// TwinCAT 3 PLC project PLC
// ProgramVersion: 3.1.4024.0
// libraries:
//   EfficientIO Communicator, * (EfficientIO)
//   EfficientIO Energy Basic, * (EfficientIO)
//   Lynus Energy ModbusRTU, * (Lynus AG)
//   Lynus HTTP Functions, * (Lynus AG)
//   Lynus Persistent Data V1, * (Lynus AG)
//   Lynus Standards, * (EfficientIO)
//   Tc2_Math, * (Beckhoff Automation GmbH)
//   Tc2_MBus, * (Beckhoff Automation GmbH)
//   Tc2_ModbusRTU, * (Beckhoff Automation GmbH)
//   Tc2_SerialCom, * (Beckhoff Automation GmbH)
//   Tc2_Standard, * (Beckhoff Automation GmbH)
//   Tc2_System, * (Beckhoff Automation GmbH)
//   Tc2_TcpIp, * (Beckhoff Automation GmbH)
//   Tc2_Utilities, * (Beckhoff Automation GmbH)
//   Tc3_IotBase, * (Beckhoff Automation GmbH)
//   Tc3_JsonXml, * (Beckhoff Automation GmbH)
//   Tc3_Module, * (Beckhoff Automation GmbH)
//   VModbusBase, * (VSA GmbH)
//   VModbusTcp, * (VSA GmbH)
// project tree:
//   / FastTask.TcTTO, MiddleTask.TcTTO, SlowTask.TcTTO
//   FB/ FB_Delta_PV_Inverter_Sunspec.TcPOU (not stored) (excluded from build), FB_Hoval.TcPOU, FB_KL6xxx_ModbusRTU_22B_Master.TcPOU (excluded from build), FB_ShellyHT_Udp.TcPOU, FB_Shelly_3EM.TcPOU (not stored) (excluded from build), FB_Shelly_HT.TcPOU (excluded from build), FB_Shelly_3EM_Helper.TcPOU (not stored) (excluded from build), FB_Shelly_HTplus.TcPOU (excluded from build), FB_Shelly_HT_Helper.TcPOU (not stored) (excluded from build), FB_Shelly_HTplus_Helper.TcPOU (excluded from build), FB_Shelly_Pro.TcPOU (excluded from build), FB_Shelly_Pro3EM.TcPOU, FB_Shelly_Pro3EM_Helper.TcPOU (not stored)
//   POUs/ prgComEffIO.TcPOU, prgEM.TcPOU, prgGrid.TcPOU (not stored), prgHeizen.TcPOU, prgHouse.TcPOU, prgMBUS.TcPOU, prgPersistent.TcPOU, prgPV.TcPOU, prgRWEffIO.TcPOU (not stored), prgSmartMe.TcPOU, prgVarEffIO.TcPOU (not stored)
// real-time tasks:
//   TASK FastTask: cycle T#5ms, priority 19, ADS port 351
//   TASK SlowTask: cycle T#20ms, priority 21, ADS port 352
//   TASK MiddleTask: cycle T#10ms, priority 20, ADS port 353
// I/O:
//   DEVICE Gerät 2 (CX-BK)
//     Box 1 (CX-BK)
//   DEVICE Device 1 (Beckhoff CCAT)
//   DEVICE Device 3 (RT-Ethernet Protocol), AmsNetId 5.123.218.205.4.1
//     Box 2 (BK9050)
// variable links:
//   PLC/PLC Instance <-> Device 2 (CX-BK)/Box 1 (CX-BK)
//     FastTask Inputs/prgMBUS.stComIn @bit {16..184 step 8} <-> Term 2 (KL6781)/Channel 1/Data In {0..21}  (22 links)
//     FastTask Inputs/prgMBUS.stComIn <-> Term 2 (KL6781)/Channel 1/Status
//     FastTask Outputs/prgMBUS.stComOut <-> Term 2 (KL6781)/Channel 1/Ctrl
//     FastTask Outputs/prgMBUS.stComOut @bit {16..184 step 8} <-> Term 2 (KL6781)/Channel 1/Data Out {0..21}  (22 links)
//     MiddleTask Inputs/prgGrid.fbGrid.fbKL3403.byStateCH1 <-> Term 5 (KL3403)/Channel 1/Status
//     MiddleTask Inputs/prgGrid.fbGrid.fbKL3403.byStateCH2 <-> Term 5 (KL3403)/Channel 2/Status
//     MiddleTask Inputs/prgGrid.fbGrid.fbKL3403.byStateCH3 <-> Term 5 (KL3403)/Channel 3/Status
//     MiddleTask Inputs/prgGrid.fbGrid.fbKL3403.iDataInCH1 <-> Term 5 (KL3403)/Channel 1/Daten Ein
//     MiddleTask Inputs/prgGrid.fbGrid.fbKL3403.iDataInCH2 <-> Term 5 (KL3403)/Channel 2/Daten Ein
//     MiddleTask Inputs/prgGrid.fbGrid.fbKL3403.iDataInCH3 <-> Term 5 (KL3403)/Channel 3/Daten Ein
//     MiddleTask Inputs/prgGrid.fbKBusState.uiKBusState_OUT <-> Inputs/State
//     MiddleTask Outputs/prgGrid.fbGrid.fbKL3403.byCntrCH1 <-> Term 5 (KL3403)/Channel 1/Kontrolle
//     MiddleTask Outputs/prgGrid.fbGrid.fbKL3403.byCntrCH2 <-> Term 5 (KL3403)/Channel 2/Kontrolle
//     MiddleTask Outputs/prgGrid.fbGrid.fbKL3403.byCntrCH3 <-> Term 5 (KL3403)/Channel 3/Kontrolle
//   PLC/PLC Instance <-> Device 3 (RT-Ethernet Protocol)/Box 2 (BK9050)
//     FastTask Inputs/prgPV.fb_RTU_Master.fbmodbusmaster.InData @bit {16..184 step 8} <-> Term 4 (KL6041)/Channel 1/Data In {0..21}  (22 links)
//     FastTask Inputs/prgPV.fb_RTU_Master.fbmodbusmaster.InData <-> Term 4 (KL6041)/Channel 1/State
//     FastTask Outputs/prgPV.fb_RTU_Master.fbmodbusmaster.OutData <-> Term 4 (KL6041)/Channel 1/Ctrl
//     FastTask Outputs/prgPV.fb_RTU_Master.fbmodbusmaster.OutData @bit {16..184 step 8} <-> Term 4 (KL6041)/Channel 1/Data Out {0..21}  (22 links)

CONFIGURATION PLC
    RESOURCE PLC ON TwinCAT3
        TASK FastTask(INTERVAL := T#5ms, PRIORITY := 19);
        TASK MiddleTask(INTERVAL := T#10ms, PRIORITY := 20);
        TASK SlowTask(INTERVAL := T#20ms, PRIORITY := 21);
        PROGRAM prgRWEffIO WITH FastTask : prgRWEffIO;
        PROGRAM prgVarEffIO WITH FastTask : prgVarEffIO;
        PROGRAM prgPV WITH FastTask : prgPV;
        PROGRAM prgMBUS WITH FastTask : prgMBUS;
        PROGRAM prgPersistent WITH MiddleTask : prgPersistent;
        PROGRAM prgGrid WITH MiddleTask : prgGrid;
        PROGRAM prgHouse WITH MiddleTask : prgHouse;
        PROGRAM prgEM WITH MiddleTask : prgEM;
        PROGRAM prgSmartMe WITH MiddleTask : prgSmartMe;
        PROGRAM prgHeizen WITH MiddleTask : prgHeizen;
        PROGRAM prgComEffIO WITH SlowTask : prgComEffIO;
    END_RESOURCE
END_CONFIGURATION

// ---- POUs/prgPV.TcPOU
PROGRAM prgPV
VAR
	lrPower_PV1					: LREAL;								//{#lynus.ag#()}
	lrPower_PV2					: LREAL;								//{#lynus.ag#()}
	lrPower_PV3					: LREAL;								//{#lynus.ag#()}
	fb_PV_1						: FB_delta_PV_inverter_sunspec;
	fb_PV_2						: FB_delta_PV_inverter_sunspec;
	fb_PV_3						: FB_delta_PV_inverter_sunspec;

	fb_RTU_Master 				: FB_KL6xxx_ModbusRTU_22B_Master;
	fbModbusRtuMaster_KL6x22B	: ModbusRtuMaster_KL6x22B;
	uint_KBusState				: UINT;							//{#lynus.ag#()}
	fbConfigKL6041 				: KL6Configuration;
	mExecute					: BOOL:= FALSE;
	int_Handshake				: INT:=0;
	mode						: ComSerialLineMode_t:=2;	
	wArrayReceiveBuffer			: ARRAY[0..130] OF WORD;
	lrCounterPV1				: LREAL;				//{#lynus.ag#()}
	lrCounterPV2				: LREAL;				//{#lynus.ag#()}
	lrCounterPV3				: LREAL;				//{#lynus.ag#()}
	rHeatSinkTemp_PV1			: REAL;					//{#lynus.ag#()}
	rHeatSinkTemp_PV2			: REAL;					//{#lynus.ag#()}
	rHeatSinkTemp_PV3			: REAL;					//{#lynus.ag#()}
	rCabinetTemp_PV1			: REAL;					//{#lynus.ag#()}
	rCabinetTemp_PV2			: REAL;					//{#lynus.ag#()}
	rCabinetTemp_PV3			: REAL;					//{#lynus.ag#()}
	usiAddress					: BYTE;
	usi_ScannedAddress			: REAL;
	
END_VAR


fb_RTU_Master(
	bConfigTerminal:= TRUE, 
	uiKBusState_IN:= uint_KBusState, 
	bBusy=> , 
	byErrorWarning=> , 
	byActualAdressInUse=> , 
	diNrOfMBRTUMasterLine_OUT=> , 
	eMessageMBRTUMaster=> , 
	bTerminalIsConfigured=> );

fb_PV_1(
	bEnable:= TRUE, 
	byMBAdress:=2 , 
	diNrOfMBRTUMasterLine_IN:= fb_RTU_Master.diNrOfMBRTUMasterLine_OUT, 
	stDeltaInverterData=> , 
	stDataEMPower_PV=> , 
	stDataEMCounter_PV=> , 
	diNrOfEM_OUT_PV=> );
fb_PV_2(
	bEnable:= TRUE, 
	byMBAdress:=3 , 
	diNrOfMBRTUMasterLine_IN:= fb_RTU_Master.diNrOfMBRTUMasterLine_OUT, 
	stDeltaInverterData=> , 
	stDataEMPower_PV=> , 
	stDataEMCounter_PV=> , 
	diNrOfEM_OUT_PV=> );
fb_PV_3(
	bEnable:= true, 
	byMBAdress:=4 , 
	diNrOfMBRTUMasterLine_IN:= fb_RTU_Master.diNrOfMBRTUMasterLine_OUT, 
	stDeltaInverterData=> , 
	stDataEMPower_PV=> , 
	stDataEMCounter_PV=> , 
	diNrOfEM_OUT_PV=> );
lrPower_PV1 		:=fb_PV_1.stDataEMPower_PV.lrPowerTotal;
lrPower_PV2 		:=fb_PV_2.stDataEMPower_PV.lrPowerTotal;
lrPower_PV3 		:=fb_PV_3.stDataEMPower_PV.lrPowerTotal;
lrCounterPV1 		:= fb_PV_1.stDataEMCounter_PV.lrCounterEnergyT1_Production;
lrCounterPV2 		:= fb_PV_2.stDataEMCounter_PV.lrCounterEnergyT1_Production;
lrCounterPV3 		:= fb_PV_3.stDataEMCounter_PV.lrCounterEnergyT1_Production;
rHeatSinkTemp_PV1	:= fb_PV_1.stDeltaInverterData.rHeatSinkTemp;
rHeatSinkTemp_PV2	:= fb_PV_2.stDeltaInverterData.rHeatSinkTemp;
rHeatSinkTemp_PV3	:= fb_PV_3.stDeltaInverterData.rHeatSinkTemp;
rCabinetTemp_PV1	:= fb_PV_1.stDeltaInverterData.rCabinetTemp;
rCabinetTemp_PV2	:= fb_PV_2.stDeltaInverterData.rCabinetTemp;
rCabinetTemp_PV3	:= fb_PV_3.stDeltaInverterData.rCabinetTemp;

(*
fbModbusRtuMaster_KL6x22B.ReadRegs(
	UnitID		:=2,
	Quantity	:=10,
	MBAddr		:=0,
	cbLength	:=20,
	pMemoryAddr	:= ADR(wArrayReceiveBuffer),
	Execute		:= TRUE,
	Timeout		:=t#1s,
	BUSY		=>,
	Error		=>,
	ErrorId		=>,
	cbRead		=>
);


fbModbusRtuMaster_KL6x22B.Execute := FALSE;

FOR usiAddress := 1 TO 247 DO
   fbModbusRtuMaster_KL6x22B.ReadRegs(UnitID := usiAddress, Execute := TRUE);
   IF NOT fbModbusRtuMaster_KL6x22B.Error THEN
      usi_ScannedAddress := usiAddress;
      EXIT;
   END_IF;
END_FOR;


// necessary for KL6041 to write the com settings
fbConfigKL6041(
	Execute 		:= mExecute,
	Mode 			:= mode,
	Baudrate 		:= 19200,
	NoDatabits 		:= 8,
	Parity 			:= 0,
	Stopbits 		:= 1,
	Handshake  		:= RS485_HALFDUPLEX, //int_Handshake,
	ContinousMode 	:= FALSE,
	pComIn 			:= ADR(fbModbusRtuMaster_KL6x22B.InData),
	pComOut 		:= ADR(fbModbusRtuMaster_KL6x22B.OutData),
	SizeComIn 		:= SIZEOF(fbModbusRtuMaster_KL6x22B.InData)		//fbModbusRtuMaster_KL6x22B
); *)

END_PROGRAM

// ---- FB/FB_KL6xxx_ModbusRTU_22B_Master.TcPOU
FUNCTION_BLOCK FB_KL6xxx_ModbusRTU_22B_Master
VAR_INPUT
	bConfigTerminal							: BOOL;																		//Possibility to configure the Terminal manually (Its only possible when the Terminal is not configured successfully)
	uiKBusState_IN							: UINT;																		//K-Bus State from the K-Bus Box on wich the Terminal is connected. (Connect with FB_K_Bus_state)
END_VAR
VAR_OUTPUT
	bBusy									: BOOL;																		//Function is Busy
	byErrorWarning							: BYTE;																		//Error Warning State
	byActualAdressInUse						: BYTE;																		//Actual Modbus Adress in Use
	diNrOfMBRTUMasterLine_OUT				: DINT;																		//Active Number from the RTU Master Function for using on other functions
	eMessageMBRTUMaster						: E_Message_MBRTUMaster;													//Message from the RTU Master Function
END_VAR				
VAR_OUTPUT PERSISTENT
	bTerminalIsConfigured					: BOOL;																		//Its True when the configuration is successfully
END_VAR
VAR		
	config_execute							: BOOL ;
	//{attribute 'hide'}
	fbKL6xxxConfig							: KL6configuration;															//FB KL6xxx to config the terminal
	fbmodbusmaster							: ModbusRtuMaster_KL6x22B;													//FB Modbus RTU
	{attribute 'hide'}
	fbmodbusmaster_Init						: ModbusRtuMaster_KL6x22B;													//FB Modbus RTU Master for workaroud regarding the internal Beckhoff problem in this function
	{attribute 'hide'}
	fbNumberDevice							: FB_NumberOfDevice;														//Function block to calcualte the number of the Device	
	{attribute 'hide'}
	fbModbusRTUMessage						: FB_MBRTUMaster_Messages;													//Modbus RTU Messages	
	{attribute 'hide'}
	FPConfigManual							: R_TRIG;																	//Internal positive Edge
	{attribute 'hide'}
	FPConfigAuto							: R_TRIG;																	//Internal positive Edge
	{attribute 'hide'}
	FPProcessCompleted						: R_TRIG;																	//Internal positive Edge
	{attribute 'hide'}
	FPError									: R_TRIG;																	//Internal positive Edge
	{attribute 'hide'}
	FPErrorIsActive							: R_TRIG;																	//Internal positive Edge
	{attribute 'hide'}
	FNInitSmall								: F_TRIG;																	//Internal negative Edge
	{attribute 'hide'}
	FNBusy									: F_TRIG;																	//Internal negative Edge
	{attribute 'hide'}
	timInit									: TON;																		//Delay to start the Terminal Configuration after the start from the plc
	{attribute 'hide'}
	timTimout								: TON;																		//Timer Timout to go on next Modbus Adress when the Ack is not set back to False
	{attribute 'hide'}
	timDissableFunctions					: TON;																		//Timer to dissable the Function after Lynus_Standards.Constants_General.tTimeDissableLynusFunctions Days without connection to the Lynus Cloud
	{attribute 'hide'}
	timResetConnectionOnGVL					: TON;																		//Timer to try reset the connection Flag on the GVL. (When somebody delete the Connection Function and make only a onlinechange)
	{attribute 'hide'}
	arrPD									: ARRAY[1..2] OF FB_PersistentData_Number;									//Function to save persistent data
	{attribute 'hide'}
	bTakeActualAdress						: BOOL;																		//True if the Current address is to be used
	{attribute 'hide'}
	bAdressHasChanged						: BOOL;																		//True if the Adress has changed
	{attribute 'hide'}
	bErrorIsActive							: BOOL;																		//True if a Error is happend. False after the next successfully read or write command
	{attribute 'hide'}
	bStopReadWrite							: BOOL;																		//Stop Function because Modbus Adress has chaged
	{attribute 'hide'}
	byLPSmallestAdress						: BYTE;																		//Loop to find out the smallest Modbus Adress
	{attribute 'hide'}
	byLPBiggestAdress						: BYTE;																		//Loop to find out the biggest Modbus Adress
	{attribute 'hide'}
	byLPActualAdress						: BYTE;																		//Loop to find out the next actuall adress
	{attribute 'hide'}
	byLPNumbersOfTotalSlaves				: BYTE;																		//Loop to find out the number of total Modbus Slaves
	{attribute 'hide'}
	bySmallestAdress						: BYTE;																		//Smallest Modbus Adress
	{attribute 'hide'}
	byBiggestAdress							: BYTE;																		//Biggest Modbus Adress
	{attribute 'hide'}
	byActualAdressInUse_CP					: BYTE;																		//Actual Modbus Adress in Use to compare it with the old one
	{attribute 'hide'}
	byNumberOfTotalSlaves					: BYTE;																		//Number of all Modbus Slaves
	{attribute 'hide'}
	byWaitInStep							: BYTE;																		//Wait in Step before start to clean data on PLC
	{attribute 'hide'}
	byLPMBAdress							: BYTE;																		//Loop for manage new Modbus Adress List after a change
	{attribute 'hide'}
	bySearchMBAdress						: BYTE;																		//Search Modbus Adress after change
	{attribute 'hide'}
	byPosInArrayMBAdress					: BYTE;																		//Save new Range from Modbus adress in the Array after a change
	{attribute 'hide'}
	iStateGVLData							: INT;																		//State machine to handle the data on the GVL
	{attribute 'hide'}
	iStateSetMBAdress						: INT;																		//State machin eto order the Modbus Adress after a change
	{attribute 'hide'}
	diCounterForGVL							: DINT;																		//Counter to clean old data on GVL
	{attribute 'hide'}
	arrRead									: ARRAY[1..Constants_Bussystems.wQuantityOfRegistersMBRTUMaster] OF WORD;	//Puffer for read out data
	{attribute 'hide'}
	arrMBAdress								: ARRAY[1..247] OF BYTE;													//Array with the actual Modbus Adress Config
END_VAR
VAR PERSISTENT
	{attribute 'conditionalshow'}
	eDeviceType								: E_MBRTUMaster_DeviceType;													//Device Type on witch the Terminal is configured
END_VAR

//Creator : Kai Ebensperger
//Company : Lynus AG
//Date : 08.07.2021
//Version : 1.0.0.0

//With this FB a serial 22 byte terminal can be configured and data can be sent/received via Modbus RTU.
//Only devices of the same type may be operated on the same master (because its not good to write to much new configurations on the terminal).
//The 1 slave that is called before the master FB in the PLC code configures the terminal
//The block must be called in a task of 5MS
//The system works according to the Master Slave principle
//Multiple communication is not possible in RTU principle

//NOTE for diNr.....Designation => 
//_IN = Here Data come in from other Functions or go out to other functions about the GVL
//_OUT = Here Data go out to other functions about the GVL

(*-------------------------------------------------------------Calcualte the number of RTU Master---------------------------------------------------------------*)

fbNumberDevice(
	diActualNumberOfDevices:= Lynus_Standards.GVL_Bussystems.diNumberOfMBRTUMasters, 
	diMaxNumberOfDevices:= Constants_Bussystems.diMaxNumberOfMBRTUMasterKL6xxx, 
	udiCounterOnlineChange:= TwinCAT_SystemInfoVarList._AppInfo.OnlineChangeCnt, 
	bNumberIsCalculatet=> , 
	bFPNumberIsCalculatet=> , 
	bOnlineChange=> , 
	diNumberForThisDevice=> diNrOfMBRTUMasterLine_OUT, 
	diNumberOfTotalDevices=> );

//Write new Numer on GVL
IF fbNumberDevice.bFPNumberIsCalculatet THEN
	Lynus_Standards.GVL_Bussystems.diNumberOfMBRTUMasters := fbNumberDevice.diNumberOfTotalDevices;	
END_IF 

//Delete old Number on GVL
IF fbNumberDevice.bOnlineChange THEN 
	Lynus_Standards.GVL_Bussystems.diNumberOfMBRTUMasters := diNrOfMBRTUMasterLine_OUT;	
		iStateGVLData := 1; 
END_IF	
	
(*-------------------------------------------------------------Service from Backend is ready and check the connection to backen for dissabel/enable Function---------------------------------------------------------------*)

//Try to reset the variable for connection on the GVL. When all is normal then the Lynus Mqtt connection function set this variable to true in the next cycle
//When we have no connection to the backend then after Lynus_Standards.Constants_General.tTimeDissableLynusFunctions days the Function is dissabled with all of his functionalities
timResetConnectionOnGVL(IN:= NOT timResetConnectionOnGVL.Q, PT:= T#1H, Q=> , ET=> );
	IF timResetConnectionOnGVL.Q THEN Lynus_Standards.GVL_Communicator.bStateConnectionToEnableFunctions := FALSE; END_IF
		IF NOT Lynus_Standards.GVL_Communicator.bStateConnectionToEnableFunctions THEN timDissableFunctions.IN := TRUE; ELSE timDissableFunctions.IN := FALSE; END_IF  
			timDissableFunctions(IN:= , PT:= Lynus_Standards.Constants_General.tTimeDissableLynusFunctions, Q=> , ET=> );

(*------------------------------------------------------------------Configuration----------------------------------------------------------------------------*)
			
//Configurate the seriall Terminal
//The configuration is depending what Slave is connected to the terminal
timInit(IN:= Lynus_Standards.GVL_Bussystems.stDataOfMBRTUMasterKL6xxx[diNrOfMBRTUMasterLine_OUT].eMBRTUDeviceType <> E_MBRTUMaster_DeviceType.eNoModbusRTUDevice AND uiKBusState_IN = 0, PT:=T#500MS, Q=> , ET=> );

IF Lynus_Standards.GVL_Bussystems.stDataOfMBRTUMasterKL6xxx[diNrOfMBRTUMasterLine_OUT].eMBRTUDeviceType <> eDeviceType AND timInit.Q THEN
	FPConfigAuto.CLK := TRUE;
		eDeviceType := Lynus_Standards.GVL_Bussystems.stDataOfMBRTUMasterKL6xxx[diNrOfMBRTUMasterLine_OUT].eMBRTUDeviceType;
ELSE
	FPConfigAuto.CLK := FALSE;
END_IF 	 

FPConfigAuto(CLK:= , Q=> );

//Configuration from the Terminal by the Slave Type
IF Lynus_Standards.GVL_Bussystems.stDataOfMBRTUMasterKL6xxx[diNrOfMBRTUMasterLine_OUT].eMBRTUDeviceType = E_MBRTUMaster_DeviceType.ePilotPMAC201_HW THEN
	//Pilot PMAC201 HW Energymessurement Device
	fbKL6xxxConfig.Mode := SERIALLINEMODE_KL6_22B_STANDARD;
	fbKL6xxxConfig.Baudrate := 38400;
	fbKL6xxxConfig.NoDatabits := 8;
	fbKL6xxxConfig.Parity := PARITY_NONE;
	fbKL6xxxConfig.Stopbits := 1;
	fbKL6xxxConfig.Handshake := RS485_HALFDUPLEX;
	fbKL6xxxConfig.ContinousMode := FALSE;
	//Timout	
	timTimout.PT := T#2S;
	fbmodbusmaster.Timeout := T#2S;
ELSIF Lynus_Standards.GVL_Bussystems.stDataOfMBRTUMasterKL6xxx[diNrOfMBRTUMasterLine_OUT].eMBRTUDeviceType = E_MBRTUMaster_DeviceType.eDrexelAWeiss_AereosilentStratosLU_Ventilation THEN
	//Aereosilent Stratos Ventilation Drexel and Weiss
	fbKL6xxxConfig.Mode := SERIALLINEMODE_KL6_22B_STANDARD;
	fbKL6xxxConfig.Baudrate := 19200;
	fbKL6xxxConfig.NoDatabits := 8;
	fbKL6xxxConfig.Parity := PARITY_NONE;
	fbKL6xxxConfig.Stopbits := 1;
	fbKL6xxxConfig.Handshake := HANDSHAKE_NONE;
	fbKL6xxxConfig.ContinousMode := FALSE;
	//Timout	
	timTimout.PT := T#10S;
	fbmodbusmaster.Timeout := T#3S;
ELSIF Lynus_Standards.GVL_Bussystems.stDataOfMBRTUMasterKL6xxx[diNrOfMBRTUMasterLine_OUT].eMBRTUDeviceType = E_MBRTUMaster_DeviceType.eABB_CM_UFD_M31M_NAProtection THEN
	//CM_UFD_M31M ABB NA Protection
	fbKL6xxxConfig.Mode := SERIALLINEMODE_KL6_22B_STANDARD;
	fbKL6xxxConfig.Baudrate := 38400;
	fbKL6xxxConfig.NoDatabits := 8;
	fbKL6xxxConfig.Parity := PARITY_NONE;
	fbKL6xxxConfig.Stopbits := 1;
	fbKL6xxxConfig.Handshake := RS485_HALFDUPLEX;
	fbKL6xxxConfig.ContinousMode := FALSE;
	//Timout	
	timTimout.PT := T#2S;
	fbmodbusmaster.Timeout := T#1S;
ELSIF Lynus_Standards.GVL_Bussystems.stDataOfMBRTUMasterKL6xxx[diNrOfMBRTUMasterLine_OUT].eMBRTUDeviceType = E_MBRTUMaster_DeviceType.eSchrack_ECS_CIONHOME_SEMIPUBLIC THEN
	//Schrack Electric Charging Station CionHome and Semipublic
	fbKL6xxxConfig.Mode := SERIALLINEMODE_KL6_22B_STANDARD;
	fbKL6xxxConfig.Baudrate := 57600;
	fbKL6xxxConfig.NoDatabits := 8;
	fbKL6xxxConfig.Parity := PARITY_NONE;
	fbKL6xxxConfig.Stopbits := 1;
	fbKL6xxxConfig.Handshake := RS485_HALFDUPLEX;
	fbKL6xxxConfig.ContinousMode := FALSE;
	//Timout	
	timTimout.PT := T#2S;
	fbmodbusmaster.Timeout := T#2S;
ELSIF Lynus_Standards.GVL_Bussystems.stDataOfMBRTUMasterKL6xxx[diNrOfMBRTUMasterLine_OUT].eMBRTUDeviceType = E_MBRTUMaster_DeviceType.ePV_DeltaSunspec THEN
	//Delte PV Inverter with Sunspec Protocol
	fbKL6xxxConfig.Mode := SERIALLINEMODE_KL6_22B_STANDARD;
	fbKL6xxxConfig.Baudrate := 19200;
	fbKL6xxxConfig.NoDatabits := 8;
	fbKL6xxxConfig.Parity := PARITY_NONE;
	fbKL6xxxConfig.Stopbits := 1;
	fbKL6xxxConfig.Handshake := RS485_HALFDUPLEX;
	fbKL6xxxConfig.ContinousMode := FALSE;
	//Timout	
	timTimout.PT := T#2S;
	fbmodbusmaster.Timeout := T#2S;
END_IF

FPConfigManual(CLK:= bConfigTerminal, Q=> );

fbKL6xxxConfig(
	Execute := config_execute,
	//Execute:= (FPConfigAuto.Q AND NOT bTerminalIsConfigured) OR (timInit.Q AND NOT bTerminalIsConfigured AND FPConfigManual.Q), 
	Mode:= ,
	Baudrate:= , 
	NoDatabits:= , 
	Parity:= , 
	Stopbits:= , 
	Handshake:= , 
	ContinousMode:= , 
	pComIn:= ADR(fbmodbusmaster.InData), 
	pComOut:= ADR(fbmodbusmaster.OutData), 
	SizeComIn:= SIZEOF(fbmodbusmaster.InData),
	Done=> , 
	Busy=> , 
	Error=> , 
	ErrorId=> );

IF fbKL6xxxConfig.Done THEN
	bTerminalIsConfigured := TRUE;
END_IF

(*------------------------------------------------------------------Read-Write----------------------------------------------------------------------------*)
	 
//Choose the right Modbus RTU Action for Read or Write Data
IF Lynus_Standards.GVL_Bussystems.stDataOfMBRTUMasterKL6xxx[diNrOfMBRTUMasterLine_OUT].eMBRTUReadWriteMode = E_MBRTUMaster_ReadWriteMode.eModbusRTUMaster_Diagnostics THEN 
	fbmodbusmaster.Diagnostics(); 
		fbmodbusmaster.cbLength := SIZEOF(Lynus_Standards.GVL_Bussystems.stDataOfMBRTUMasterKL6xxx[diNrOfMBRTUMasterLine_OUT].arrWriteOutData);
			fbmodbusmaster.pMemoryAddr := ADR(Lynus_Standards.GVL_Bussystems.stDataOfMBRTUMasterKL6xxx[diNrOfMBRTUMasterLine_OUT].arrWriteOutData);
END_IF
IF Lynus_Standards.GVL_Bussystems.stDataOfMBRTUMasterKL6xxx[diNrOfMBRTUMasterLine_OUT].eMBRTUReadWriteMode = E_MBRTUMaster_ReadWriteMode.eModbusRTUMaster_ReadCoils THEN 
	fbmodbusmaster.ReadCoils(); 
		fbmodbusmaster.cbLength := SIZEOF(arrRead);
			fbmodbusmaster.pMemoryAddr := ADR(arrRead);	
END_IF
IF Lynus_Standards.GVL_Bussystems.stDataOfMBRTUMasterKL6xxx[diNrOfMBRTUMasterLine_OUT].eMBRTUReadWriteMode = E_MBRTUMaster_ReadWriteMode.eModbusRTUMaster_ReadInputRegs THEN 
	fbmodbusmaster.ReadInputRegs(); 
		fbmodbusmaster.cbLength := SIZEOF(arrRead);
			fbmodbusmaster.pMemoryAddr := ADR(arrRead);
END_IF
IF Lynus_Standards.GVL_Bussystems.stDataOfMBRTUMasterKL6xxx[diNrOfMBRTUMasterLine_OUT].eMBRTUReadWriteMode = E_MBRTUMaster_ReadWriteMode.eModbusRTUMaster_ReadInputStatus THEN 
	fbmodbusmaster.ReadInputStatus(); 
		fbmodbusmaster.cbLength := SIZEOF(arrRead);
			fbmodbusmaster.pMemoryAddr := ADR(arrRead);
END_IF
IF Lynus_Standards.GVL_Bussystems.stDataOfMBRTUMasterKL6xxx[diNrOfMBRTUMasterLine_OUT].eMBRTUReadWriteMode = E_MBRTUMaster_ReadWriteMode.eModbusRTUMaster_ReadRegs THEN 
	fbmodbusmaster.ReadRegs();
		fbmodbusmaster.cbLength := SIZEOF(arrRead);
			fbmodbusmaster.pMemoryAddr := ADR(arrRead); 
END_IF
IF Lynus_Standards.GVL_Bussystems.stDataOfMBRTUMasterKL6xxx[diNrOfMBRTUMasterLine_OUT].eMBRTUReadWriteMode = E_MBRTUMaster_ReadWriteMode.eModbusRTUMaster_WriteMultipleCoils THEN 
	fbmodbusmaster.WriteMultipleCoils();
		fbmodbusmaster.cbLength := SIZEOF(Lynus_Standards.GVL_Bussystems.stDataOfMBRTUMasterKL6xxx[diNrOfMBRTUMasterLine_OUT].arrWriteOutData);
			fbmodbusmaster.pMemoryAddr := ADR(Lynus_Standards.GVL_Bussystems.stDataOfMBRTUMasterKL6xxx[diNrOfMBRTUMasterLine_OUT].arrWriteOutData); 
END_IF
IF Lynus_Standards.GVL_Bussystems.stDataOfMBRTUMasterKL6xxx[diNrOfMBRTUMasterLine_OUT].eMBRTUReadWriteMode = E_MBRTUMaster_ReadWriteMode.eModbusRTUMaster_WriteRegs THEN 
	fbmodbusmaster.WriteRegs(); 
		fbmodbusmaster.cbLength := SIZEOF(Lynus_Standards.GVL_Bussystems.stDataOfMBRTUMasterKL6xxx[diNrOfMBRTUMasterLine_OUT].arrWriteOutData);
			fbmodbusmaster.pMemoryAddr := ADR(Lynus_Standards.GVL_Bussystems.stDataOfMBRTUMasterKL6xxx[diNrOfMBRTUMasterLine_OUT].arrWriteOutData);
END_IF
IF Lynus_Standards.GVL_Bussystems.stDataOfMBRTUMasterKL6xxx[diNrOfMBRTUMasterLine_OUT].eMBRTUReadWriteMode = E_MBRTUMaster_ReadWriteMode.eModbusRTUMaster_WriteSingleCoil THEN 
	fbmodbusmaster.WriteSingleCoil(); 
		fbmodbusmaster.cbLength := SIZEOF(Lynus_Standards.GVL_Bussystems.stDataOfMBRTUMasterKL6xxx[diNrOfMBRTUMasterLine_OUT].arrWriteOutData);
			fbmodbusmaster.pMemoryAddr := ADR(Lynus_Standards.GVL_Bussystems.stDataOfMBRTUMasterKL6xxx[diNrOfMBRTUMasterLine_OUT].arrWriteOutData);
END_IF
IF Lynus_Standards.GVL_Bussystems.stDataOfMBRTUMasterKL6xxx[diNrOfMBRTUMasterLine_OUT].eMBRTUReadWriteMode = E_MBRTUMaster_ReadWriteMode.eModbusRTUMaster_WriteSingleRegister THEN 
	fbmodbusmaster.WriteSingleRegister(); 
		fbmodbusmaster.cbLength := SIZEOF(Lynus_Standards.GVL_Bussystems.stDataOfMBRTUMasterKL6xxx[diNrOfMBRTUMasterLine_OUT].arrWriteOutData);
			fbmodbusmaster.pMemoryAddr := ADR(Lynus_Standards.GVL_Bussystems.stDataOfMBRTUMasterKL6xxx[diNrOfMBRTUMasterLine_OUT].arrWriteOutData);
END_IF

//Order the range of MB Adress when we have a change on that on the slave Functions
IF MEMCMP(ADR(arrMBAdress),ADR(Lynus_Standards.GVL_Bussystems.stDataOfMBRTUMasterKL6xxx[diNrOfMBRTUMasterLine_OUT].arrAllModbusSlaveAdresses),SIZEOF(Lynus_Standards.GVL_Bussystems.stDataOfMBRTUMasterKL6xxx[diNrOfMBRTUMasterLine_OUT].arrAllModbusSlaveAdresses)) <> 0 AND iStateSetMBAdress = 0 THEN
	iStateSetMBAdress := 1;
		bStopReadWrite := TRUE;
			MEMCPY(ADR(arrMBAdress),ADR(Lynus_Standards.GVL_Bussystems.stDataOfMBRTUMasterKL6xxx[diNrOfMBRTUMasterLine_OUT].arrAllModbusSlaveAdresses),SIZEOF(Lynus_Standards.GVL_Bussystems.stDataOfMBRTUMasterKL6xxx[diNrOfMBRTUMasterLine_OUT].arrAllModbusSlaveAdresses));
END_IF

CASE iStateSetMBAdress OF
	
	0://Init
		bStopReadWrite := FALSE;

	1://Set the Actual Adress in use to 0 and Clear old MB Adresses in Array
		bTakeActualAdress := FALSE;
			byActualAdressInUse := 0;
				bySearchMBAdress := 0;
					byPosInArrayMBAdress := 0;	

		FOR byLPMBAdress := 1 TO 247 BY 1 DO
			Lynus_Standards.GVL_Bussystems.stDataOfMBRTUMasterKL6xxx[diNrOfMBRTUMasterLine_OUT].arrAllModbusSlaveAdresses[byLPMBAdress] := 0;
		END_FOR 
			
			iStateSetMBAdress := 2;	
		
	2://Order the new Adresses from lowest to highest
		bySearchMBAdress := bySearchMBAdress + 1;
			bySearchMBAdress := LIMIT(1,bySearchMBAdress,247);			
	
		FOR byLPMBAdress := 1 TO 247 BY 1 DO
			IF arrMBAdress[byLPMBAdress] = bySearchMBAdress THEN
				byPosInArrayMBAdress := byPosInArrayMBAdress + 1;
					byPosInArrayMBAdress := LIMIT(1,byPosInArrayMBAdress,247);
						Lynus_Standards.GVL_Bussystems.stDataOfMBRTUMasterKL6xxx[diNrOfMBRTUMasterLine_OUT].arrAllModbusSlaveAdresses[byPosInArrayMBAdress] := arrMBAdress[byLPMBAdress]; 	
			END_IF
		END_FOR  
		
		//Done
		IF bySearchMBAdress >= 247 THEN 
			iStateSetMBAdress := 0;
				MEMCPY(ADR(arrMBAdress),ADR(Lynus_Standards.GVL_Bussystems.stDataOfMBRTUMasterKL6xxx[diNrOfMBRTUMasterLine_OUT].arrAllModbusSlaveAdresses),SIZEOF(Lynus_Standards.GVL_Bussystems.stDataOfMBRTUMasterKL6xxx[diNrOfMBRTUMasterLine_OUT].arrAllModbusSlaveAdresses));
		END_IF 
	
END_CASE

//Check the Modbus Adresses from each Slave Device
FPProcessCompleted(CLK:= Lynus_Standards.GVL_Bussystems.stDataOfMBRTUMasterKL6xxx[diNrOfMBRTUMasterLine_OUT].bReadWriteIsDone, Q=> );
	FPError(CLK:= fbmodbusmaster.Error, Q=> );

bySmallestAdress := 247;	
	FOR byLPSmallestAdress := 1 TO 247 BY 1 DO
		IF Lynus_Standards.GVL_Bussystems.stDataOfMBRTUMasterKL6xxx[diNrOfMBRTUMasterLine_OUT].arrAllModbusSlaveAdresses[byLPSmallestAdress] < bySmallestAdress AND Lynus_Standards.GVL_Bussystems.stDataOfMBRTUMasterKL6xxx[diNrOfMBRTUMasterLine_OUT].arrAllModbusSlaveAdresses[byLPSmallestAdress] <> 0 THEN bySmallestAdress := Lynus_Standards.GVL_Bussystems.stDataOfMBRTUMasterKL6xxx[diNrOfMBRTUMasterLine_OUT].arrAllModbusSlaveAdresses[byLPSmallestAdress]; END_IF
	END_FOR
byBiggestAdress := 0;
	FOR byLPBiggestAdress := 1 TO 247 BY 1 DO
		IF Lynus_Standards.GVL_Bussystems.stDataOfMBRTUMasterKL6xxx[diNrOfMBRTUMasterLine_OUT].arrAllModbusSlaveAdresses[byLPBiggestAdress] > byBiggestAdress THEN byBiggestAdress := Lynus_Standards.GVL_Bussystems.stDataOfMBRTUMasterKL6xxx[diNrOfMBRTUMasterLine_OUT].arrAllModbusSlaveAdresses[byLPBiggestAdress]; END_IF  
	END_FOR
//Take the Next Adress after the Read/write is done
IF FPProcessCompleted.Q OR FPError.Q THEN
	bTakeActualAdress := TRUE;
		FOR byLPActualAdress := 1 TO 247 BY 1 DO
			IF Lynus_Standards.GVL_Bussystems.stDataOfMBRTUMasterKL6xxx[diNrOfMBRTUMasterLine_OUT].arrAllModbusSlaveAdresses[byLPActualAdress] > byActualAdressInUse THEN 
				byActualAdressInUse := Lynus_Standards.GVL_Bussystems.stDataOfMBRTUMasterKL6xxx[diNrOfMBRTUMasterLine_OUT].arrAllModbusSlaveAdresses[byLPActualAdress]; 
					EXIT;
			END_IF
		END_FOR		
END_IF

//Count the Number of RTU Slaves
byNumberOfTotalSlaves := 0;
	FOR byLPNumbersOfTotalSlaves := 1 TO 247 BY 1 DO
		IF Lynus_Standards.GVL_Bussystems.stDataOfMBRTUMasterKL6xxx[diNrOfMBRTUMasterLine_OUT].arrAllModbusSlaveAdresses[byLPNumbersOfTotalSlaves] <> 0 THEN byNumberOfTotalSlaves := byNumberOfTotalSlaves + 1; END_IF
	END_FOR

FNInitSmall(CLK:= bySmallestAdress = 247, Q=> );

IF byActualAdressInUse <> byActualAdressInUse_CP THEN bAdressHasChanged := TRUE; byActualAdressInUse_CP := byActualAdressInUse; ELSE bAdressHasChanged := FALSE; END_IF 

IF ((FPError.Q OR FPProcessCompleted.Q) AND NOT bAdressHasChanged) OR FNInitSmall.Q OR bySmallestAdress = byBiggestAdress THEN byActualAdressInUse := bySmallestAdress; END_IF

timTimout(IN:= Lynus_Standards.GVL_Bussystems.stDataOfMBRTUMasterKL6xxx[diNrOfMBRTUMasterLine_OUT].bReadWriteIsDone, PT:= , Q=> , ET=> );

IF FPProcessCompleted.Q OR timTimout.Q THEN Lynus_Standards.GVL_Bussystems.stDataOfMBRTUMasterKL6xxx[diNrOfMBRTUMasterLine_OUT].bReadWriteIsDone := FALSE; END_IF

IF NOT bTakeActualAdress THEN 
	fbmodbusmaster.UnitID := bySmallestAdress;
ELSE
	fbmodbusmaster.UnitID := byActualAdressInUse;
END_IF

fbmodbusmaster(
	UnitID:= , 
	Quantity:= Lynus_Standards.GVL_Bussystems.stDataOfMBRTUMasterKL6xxx[diNrOfMBRTUMasterLine_OUT].wNumberOfRegister, 
	MBAddr:= Lynus_Standards.GVL_Bussystems.stDataOfMBRTUMasterKL6xxx[diNrOfMBRTUMasterLine_OUT].wModbusRegister, 
	cbLength:= , 
	pMemoryAddr:= , 
	Execute:= Lynus_Standards.GVL_Bussystems.stDataOfMBRTUMasterKL6xxx[diNrOfMBRTUMasterLine_OUT].bSlaveStartReadOrWrite AND bTerminalIsConfigured AND NOT timDissableFunctions.Q AND NOT bStopReadWrite, 
	Timeout:= , 
	BUSY=> , 
	Error=> , 
	ErrorId=> , 
	cbRead=> );	
	
(*------------------------------------------------------------------Busy Flag----------------------------------------------------------------------------*)

IF NOT bTerminalIsConfigured THEN
	bBusy := fbKL6xxxConfig.Busy;
ELSE
	bBusy := fbmodbusmaster.BUSY;
END_IF

//When we have a change on the MB Adress List we set the Function always on Busy that al other Slave Functions Stops in the Init Step
IF bStopReadWrite THEN bBusy := TRUE; END_IF

FNBusy(CLK:= fbmodbusmaster.BUSY, Q=> );

(*------------------------------------------------------------------Error and Warning----------------------------------------------------------------------------*)

IF timDissableFunctions.Q THEN fbModbusRTUMessage.bWarning := TRUE; fbModbusRTUMessage.iWarningCode := 0; ELSE fbModbusRTUMessage.bWarning := FALSE; END_IF   
	IF (Lynus_Standards.GVL_Bussystems.diNumberOfMBRTUMasters > Constants_Bussystems.diMaxNumberOfMBRTUMasterKL6xxx) OR (NOT bTerminalIsConfigured AND fbKL6xxxConfig.Error) OR (bTerminalIsConfigured AND fbmodbusmaster.Error) OR bStopReadWrite THEN 
		fbModbusRTUMessage.bError := TRUE;
	ELSE
		fbModbusRTUMessage.bError := FALSE;
	END_IF

IF Lynus_Standards.GVL_Bussystems.diNumberOfMBRTUMasters > Constants_Bussystems.diMaxNumberOfMBRTUMasterKL6xxx THEN
	fbModbusRTUMessage.iErrorCode := 1;	
ELSIF NOT bTerminalIsConfigured THEN 
	IF fbKL6xxxConfig.Error THEN 
		fbModbusRTUMessage.iErrorCode := 2; 
	END_IF
//When we have a change on the MB Adress List we set the Function always on Error that al other Slave Functions go back to the Init Step
ELSIF bStopReadWrite THEN
	fbModbusRTUMessage.iErrorCode := 2; 
ELSE
	IF fbmodbusmaster.ErrorId = 1 THEN fbModbusRTUMessage.iErrorCode := 3; END_IF
	IF fbmodbusmaster.ErrorId = 2 THEN fbModbusRTUMessage.iErrorCode := 4; END_IF
	IF fbmodbusmaster.ErrorId = 3 THEN fbModbusRTUMessage.iErrorCode := 5; END_IF
	IF fbmodbusmaster.ErrorId = 4 THEN fbModbusRTUMessage.iErrorCode := 6; END_IF
	IF fbmodbusmaster.ErrorId = 5 THEN fbModbusRTUMessage.iErrorCode := 7; END_IF
	IF fbmodbusmaster.ErrorId = 6 THEN fbModbusRTUMessage.iErrorCode := 8; END_IF
	IF fbmodbusmaster.ErrorId = 7 THEN fbModbusRTUMessage.iErrorCode := 9; END_IF
	IF fbmodbusmaster.ErrorId = 8 THEN fbModbusRTUMessage.iErrorCode := 10; END_IF
	IF fbmodbusmaster.ErrorId = 16#A THEN fbModbusRTUMessage.iErrorCode := 11; END_IF
	IF fbmodbusmaster.ErrorId = 16#B THEN fbModbusRTUMessage.iErrorCode := 12; END_IF
	IF fbmodbusmaster.ErrorId = 16#20 THEN fbModbusRTUMessage.iErrorCode := 13; END_IF
	IF fbmodbusmaster.ErrorId = 16#21 THEN fbModbusRTUMessage.iErrorCode := 14; END_IF
	IF fbmodbusmaster.ErrorId = 16#22 THEN fbModbusRTUMessage.iErrorCode := 15; END_IF
	IF fbmodbusmaster.ErrorId = 16#23 THEN fbModbusRTUMessage.iErrorCode := 16; END_IF
	IF fbmodbusmaster.ErrorId = 16#24 THEN fbModbusRTUMessage.iErrorCode := 17; END_IF
	IF fbmodbusmaster.ErrorId = 16#25 THEN fbModbusRTUMessage.iErrorCode := 18; END_IF
	IF fbmodbusmaster.ErrorId = 102 THEN fbModbusRTUMessage.iErrorCode := 19; END_IF
	IF fbmodbusmaster.ErrorId = 103 THEN fbModbusRTUMessage.iErrorCode := 20; END_IF
	IF fbmodbusmaster.ErrorId = 107 THEN fbModbusRTUMessage.iErrorCode := 21; END_IF
	IF fbmodbusmaster.ErrorId = 110 THEN fbModbusRTUMessage.iErrorCode := 22; END_IF
	IF fbmodbusmaster.ErrorId = 120 THEN fbModbusRTUMessage.iErrorCode := 23; END_IF
	IF fbmodbusmaster.ErrorId = 150 THEN fbModbusRTUMessage.iErrorCode := 24; END_IF
	IF fbmodbusmaster.ErrorId = 232 THEN fbModbusRTUMessage.iErrorCode := 25; END_IF
	IF fbmodbusmaster.ErrorId = 233 THEN fbModbusRTUMessage.iErrorCode := 26; END_IF
END_IF

fbModbusRTUMessage(
	bTerminalConfigured:= bTerminalIsConfigured, 
	bError:= , 
	bWarning:= , 
	iWarningCode:= , 
	iErrorCode:= , 
	byErrorWarning=> byErrorWarning, 
	eMessageMBRTUMaster=> eMessageMBRTUMaster);

//Set this Flag after a Error and Reset after next Read or Write command without Error	
IF FPError.Q THEN bErrorIsActive := TRUE; END_IF
	IF FNBusy.Q AND NOT fbmodbusmaster.Error THEN bErrorIsActive := FALSE; END_IF	
	
FPErrorIsActive(CLK:= bErrorIsActive, Q=> );
	
(*-----------------------------------------------------------Handle data to Global structure for Modbus RTU Communication-----------------------------------------------------------------*)

CASE iStateGVLData OF
	
	0://Init Step
		byWaitInStep := 0;
			diCounterForGVL := 1;
	
	1://Wait for 4 Steps before clean al Data on GVL
		byWaitInStep := byWaitInStep + 1;
			IF byWaitInStep >= 4 AND fbNumberDevice.bNumberIsCalculatet THEN iStateGVLData := 2; END_IF
				//To much Devices, back to the Init step
				IF byWaitInStep >= 4 AND NOT fbNumberDevice.bNumberIsCalculatet THEN iStateGVLData := 0; END_IF	
			
	2://Clear all Data in GVL
	//Some Parts in the GVL Reset the Slave. Otherwise there will be problems when writing the new addresses to the array in the GVL.
	Lynus_Standards.GVL_Bussystems.stDataOfMBRTUMasterKL6xxx[diCounterForGVL].bMasterIsBusy := FALSE;	
		Lynus_Standards.GVL_Bussystems.stDataOfMBRTUMasterKL6xxx[diCounterForGVL].bTerminalIsConfigured := FALSE;	
			Lynus_Standards.GVL_Bussystems.stDataOfMBRTUMasterKL6xxx[diCounterForGVL].byNumberOfSlaves := 0;
				Lynus_Standards.GVL_Bussystems.stDataOfMBRTUMasterKL6xxx[diCounterForGVL].byErrorWarning := 0;
					Lynus_Standards.GVL_Bussystems.stDataOfMBRTUMasterKL6xxx[diCounterForGVL].byActualMBAdressInProgrss := 0;
						Lynus_Standards.GVL_Bussystems.stDataOfMBRTUMasterKL6xxx[diCounterForGVL].bNoNewMBusAdress := FALSE;	
														 		
		diCounterForGVL := diCounterForGVL + 1;
			diCounterForGVL := LIMIT(0,diCounterForGVL,Constants_Bussystems.diMaxNumberOfMBRTUMasterKL6xxx);
				//Back to the init step
				IF diCounterForGVL >= Constants_Bussystems.diMaxNumberOfMBRTUMasterKL6xxx THEN iStateGVLData := 0; END_IF

END_CASE 
	
IF diNrOfMBRTUMasterLine_OUT > 0 AND fbNumberDevice.bNumberIsCalculatet THEN  
	Lynus_Standards.GVL_Bussystems.stDataOfMBRTUMasterKL6xxx[diNrOfMBRTUMasterLine_OUT].bMasterIsBusy := bBusy;
		Lynus_Standards.GVL_Bussystems.stDataOfMBRTUMasterKL6xxx[diNrOfMBRTUMasterLine_OUT].byErrorWarning := byErrorWarning;
			Lynus_Standards.GVL_Bussystems.stDataOfMBRTUMasterKL6xxx[diNrOfMBRTUMasterLine_OUT].bTerminalIsConfigured := bTerminalIsConfigured;
				Lynus_Standards.GVL_Bussystems.stDataOfMBRTUMasterKL6xxx[diNrOfMBRTUMasterLine_OUT].byActualMBAdressInProgrss := fbmodbusmaster.UnitID;
					Lynus_Standards.GVL_Bussystems.stDataOfMBRTUMasterKL6xxx[diNrOfMBRTUMasterLine_OUT].byNumberOfSlaves := byNumberOfTotalSlaves;
						Lynus_Standards.GVL_Bussystems.stDataOfMBRTUMasterKL6xxx[diCounterForGVL].bNoNewMBusAdress := bStopReadWrite;
						IF FNBusy.Q THEN
							IF NOT fbmodbusmaster.Error THEN
								Lynus_Standards.GVL_Bussystems.stDataOfMBRTUMasterKL6xxx[diNrOfMBRTUMasterLine_OUT].arrReadOutData := arrRead;
							ELSE
								//Workarround about internal Beckhoff Lib Error 
								IF FPErrorIsActive.Q THEN 
									MEMCPY(ADR(fbmodbusmaster),ADR(fbmodbusmaster_Init),SIZEOF(fbmodbusmaster_Init));
								END_IF
							END_IF
						END_IF	
END_IF	
	
(*----------------------------------------------------------Save persistent data----------------------------------------------------------------*)

arrPD[1](lrValue:= BOOL_TO_LREAL(bTerminalIsConfigured), bEventBasedActive=> );
arrPD[2](lrValue:= INT_TO_LREAL(eDeviceType), bEventBasedActive=> );

END_FUNCTION_BLOCK

// ---- POUs/prgMBUS.TcPOU
PROGRAM prgMBUS
VAR
	// M-Bus Kommunikation (KL6781)
	fbMBusKL6781    : FB_MBUSKL6781;             // Hauptbaustein für die M-Bus-Kommunikation
	stComIn  AT %I* : ST_KL6781inData22B; // Eingabestruktur für KL6781
	stComOut AT %Q* : ST_KL6781outData22B;// Ausgabestruktur für KL6781
	stCom           : ST_MBUS_Communication;     // Kommunikationsstruktur für alle M-Bus-Geräte
	fbScann         : FB_MBUS_Scan;

	fbWaermeGesamt     : FB_MBUS_General:= (bStart:= TRUE);          	 // Funktionsbaustein für Holzkessel
  	eWaermeGesamtErr   : E_MBUS_ERROR;  
	WaermeGesamtKWh    : LREAL;											//{#lynus.ag#()}
	WaermeGesamtKW     : LREAL;											//{#lynus.ag#()}
	

	fbMattenrainstr11  : FB_MBUS_General:= (bStart:= TRUE);          	 // Funktionsbaustein für Holzkessel
  	eMattenrainstr11Err: E_MBUS_ERROR;  
	Mattenrainstr11KWh : LREAL;											//{#lynus.ag#()}
	Mattenrainstr11KW  : LREAL;											//{#lynus.ag#()}
	
	Mattenrainstr9KWh  : LREAL;											//{#lynus.ag#()}
	Mattenrainstr9KW   : LREAL;											//{#lynus.ag#()}

END_VAR

{region "Kommunikation"}
fbMBusKL6781(
	usiRetries:= 3,                    // Anzahl der Wiederholungen bei Fehler
	bStart    := TRUE,                 // Startet die M-Bus-Kommunikation
	bDisabled := FALSE,                // Deaktiviert die M-Bus-Kommunikation nicht
	bBusy     => , 
	bReady    => , 
	bError    => , 
	eError    => , 
	stComIn  := stComIn, 
	stComOut := stComOut, 
	stCom    := stCom
);

fbScann(
	bStart:= FALSE, 
	bStop:= , 
	eBaudrate:= E_MBUS_Baudrate.eMBus_Baud2400, 
	bDisabled:= , 
	bBusy=> , 
	bReady=> , 
	bError=> , 
	eError=> , 
	usiAddress=> , 
	usiCount=> , 
	arrDevice=> , 
	stCom:= stCom);
{endregion}

{region "Wärme gesamt"}
fbWaermeGesamt(
	usiAddress:= 1,                    	// M-Bus-Adresse(Primär)
	bStart    := ,                // Startflag
	usiUnit   := 1,               		// KW
	bDisabled := , //FALSE,                 	
	bBusy     => , 
	bReady    => ,              				// Datenbereit-Status
	bError    => , 
	eError    => , 
	stCom     := stCom
);

IF NOT fbWaermeGesamt.bBusy AND fbWaermeGesamt.bError THEN

  eWaermeGesamtErr:= fbWaermeGesamt.eError;
END_IF
IF fbWaermeGesamt.bReady THEN

  eWaermeGesamtErr:= E_MBUS_ERROR.eMBus_no_error;

  WaermeGesamtKWh:= STRING_TO_REAL(fbWaermeGesamt.arrData[4].sValue);                 	// Energie (kWh)
  WaermeGesamtKW := STRING_TO_REAL(fbWaermeGesamt.arrData[9].sValue);					// Leistung (kW)
	   
END_IF
{endregion}

{region "Mattenrainstr. 11"}
fbMattenrainstr11(
	usiAddress:= 2,                    	// M-Bus-Adresse(Primär)
	bStart    := ,                // Startflag
	usiUnit   := 1,               		// KW
	bDisabled := , //FALSE,                 	
	bBusy     => , 
	bReady    => ,              				// Datenbereit-Status
	bError    => , 
	eError    => , 
	stCom     := stCom
);

IF NOT fbMattenrainstr11.bBusy AND fbMattenrainstr11.bError THEN

  eWaermeGesamtErr:= fbMattenrainstr11.eError;
END_IF
IF fbMattenrainstr11.bReady THEN

  eMattenrainstr11Err:= E_MBUS_ERROR.eMBus_no_error;

  Mattenrainstr11KWh:= STRING_TO_REAL(fbMattenrainstr11.arrData[4].sValue);                 	// Energie (kWh)
  Mattenrainstr11KW := STRING_TO_REAL(fbMattenrainstr11.arrData[9].sValue);                 	// Leistung (kW)
	   
END_IF
{endregion}

{region "Mattenrainstr. 9"} 

	 Mattenrainstr9KWh := WaermeGesamtKWh - Mattenrainstr11KWh;									// Energie (kWh)
	 Mattenrainstr9KW  := WaermeGesamtKW - Mattenrainstr11KW;									// Leistung (kW)
	 
{endregion}

END_PROGRAM

// ---- POUs/prgPersistent.TcPOU
PROGRAM prgPersistent
VAR
	fbUSV		: FB_WritePersistentData_CX81xx;
	fb_Reboot		: NT_reboot;
	m_Reboot		: BOOL:=FALSE;
END_VAR

fbUSV(
	eSaveModeData:= eUSVSaveMode.eSaveWhenPowerfail, 
	bLoadPersistentDataOk=> , 
	bPowerFailDetect=> , 
	bError=> , 
	bySaveProcess=> , 
	dwStorageLast24h=> , 
	udiErrorCode=> );
	
		
fb_Reboot(	netid := '',
			delay := 2,
			start := m_Reboot);

END_PROGRAM

// ---- POUs/prgHouse.TcPOU
PROGRAM prgHouse
VAR
	lrHousePower					: LREAL;								//{#lynus.ag#()}

END_VAR

lrHousePower := prgGrid.lrGridPower + prgPv.lrPower_PV1 + prgPv.lrPower_PV2 + prgPv.lrPower_PV3;

END_PROGRAM

// ---- POUs/prgEM.TcPOU
PROGRAM prgEM
VAR
		// Grid Objekt H 3-phase, 400V
	fb_UV_Garderobe					: FB_Shelly_Pro3EM:= (bStart:= TRUE);
	
	lrPower_UV_Garderobe_TotalkW	: LREAL;			//{#lynus.ag#()}
	lrEnergy_UV_Garderobe_Total		: LREAL;			//{#lynus.ag#()}
	lrCurrent_UV_Garderobe_L1			: LREAL;			//{#lynus.ag#()}
	lrCurrent_UV_Garderobe_L2			: LREAL;			//{#lynus.ag#()}
	lrCurrent_UV_Garderobe_L3			: LREAL;			//{#lynus.ag#()}
	lrVoltage_UV_Garderobe_L1			: LREAL;			//{#lynus.ag#()}
	lrVoltage_UV_Garderobe_L2			: LREAL;			//{#lynus.ag#()}
	lrVoltage_UV_Garderobe_L3			: LREAL;			//{#lynus.ag#()}

END_VAR

	// Grid Objekt H 3-phase, 400V
fb_UV_Garderobe(
	bStart:= , 
	tDelayRequest:= T#20S, 
	sHostname:= '172.32.12.121', 
	bValidResult=> , 
  lrpowerTotal=> lrPower_UV_Garderobe_TotalkW,
  lrpoweraprtTotal=> lrEnergy_UV_Garderobe_Total,
  lrcurrentP1=> lrCurrent_UV_Garderobe_L1,
  lrvoltageP1=> lrVoltage_UV_Garderobe_L1,
  lrcurrentP2=> lrCurrent_UV_Garderobe_L2,
  lrvoltageP2=> lrVoltage_UV_Garderobe_L2,
  lrcurrentP3=> lrCurrent_UV_Garderobe_L3,
  lrvoltageP3=> lrVoltage_UV_Garderobe_L3);

END_PROGRAM

// ---- FB/FB_Shelly_Pro3EM.TcPOU
FUNCTION_BLOCK FB_Shelly_Pro3EM
VAR_INPUT
	bStart				: BOOL;
	tDelayRequest		: TIME := T#3S;		//Timer for delay before start with the next read or write Request
	sHostname			: STRING(255);		//Hostname or IP Adress from the Server
END_VAR

VAR_IN_OUT
END_VAR

VAR_OUTPUT
	bValidResult				: BOOL;															//Valid Result received from Server
    bBusy						: BOOL;															//Function is Busy
    bError						: BOOL;															//Error sucess
	bDone						: BOOL;															//True after the decoding from the received Json File
	bConnected					: BOOL;															//Connection to the Server
	lrpowerP1					: LREAL;														//Received Value
	lrfrequencyP1				: LREAL;														//Received Value
	lrcurrentP1					: LREAL;														//Received Value
	lrvoltageP1					: LREAL;														//Received Value
	lrpowerP2					: LREAL;														//Received Value
	lrfrequencyP2				: LREAL;														//Received Value
	lrcurrentP2					: LREAL;														//Received Value
	lrvoltageP2					: LREAL;														//Received Value
	lrpowerP3					: LREAL;														//Received Value
	lrfrequencyP3				: LREAL;														//Received Value
	lrcurrentP3					: LREAL;														//Received Value
	lrvoltageP3					: LREAL;														//Received Value
	lrpowerTotal				: LREAL;														//Received Value
	lrcurrentTotal				: LREAL;														//Received Value
	lrpoweraprtTotal			: LREAL;														//Received Value
	hrErrorCode       			: HRESULT;														//Error Result from Http Client
END_VAR

VAR
	fbClient					: FB_IotHttpClient;
	fbHttpGet					: FB_Shelly_Pro3EM_Helper;
	timStartRequest				: TON;															//Timer to Start the Request
	FPStartRequest				: R_TRIG;														//Internal positive Edge
	FPDone						: R_TRIG;														//Internal positive Edge
	FNStart						: F_TRIG;														//Internal negative Edge
END_VAR

(*------------------------------------------------------------------------------------Configure HTTP Client------------------------------------------------------------------------------------------------------*)

fbClient.sHostName := sHostname;
fbClient.tConnectionTimeout := tDelayRequest;

IF NOT fbClient.bConfigured THEN 
	fbClient.nHostPort:= 80;
	fbClient.bKeepAlive := TRUE;
	fbClient.tConnectionTimeout := T#2S;
END_IF


//Timer to start the Request
FPStartRequest(CLK:= bStart, Q=> );
	timStartRequest(IN:= fbClient.bConfigured AND bStart AND NOT timStartRequest.Q, PT:= tDelayRequest, Q=> , ET=> );
		IF ((timStartRequest.Q AND NOT bBusy) OR (FPStartRequest.Q AND NOT bBusy AND fbClient.bConfigured)) THEN fbHttpGet.bSend := TRUE; END_IF

				
//Http Get Function
fbHttpGet(
(*
	lrpowerP1 => lrpowerP1,
	lrfrequencyP1 => lrfrequencyP1,
	lrcurrentP1 => lrcurrentP1,
	lrvoltageP1 => lrvoltageP1,
	lrpowerP2 => lrpowerP2,
	lrfrequencyP2 => lrfrequencyP2,
	lrcurrentP2 => lrcurrentP2,
	lrvoltageP2 => lrvoltageP2,
	lrpowerP3 => lrpowerP3,
	lrfrequencyP3 => lrfrequencyP3,
	lrcurrentP3 => lrcurrentP3,
	lr_total_current => lrcurrentTotal,
*)
  lr_a_current=> lrcurrentP1,
  lr_a_voltage=> lrvoltageP1,
  lr_b_current=> lrcurrentP2,
  lr_b_voltage=> lrvoltageP2,
  lr_c_current=> lrcurrentP3,
  lr_c_voltage=> lrvoltageP3,

	lr_total_act_power => lrpowerTotal,
	lr_total_aprt_power => lrpoweraprtTotal,
	bSend:= , 
	fbClient:= fbClient, 
	bBusy=> bBusy, 
	bError=> ,
	sContentS0=> );


fbHttpGet.bSend := FALSE;

FPDone(CLK:= bDone, Q=> );


fbClient.Execute();

//Error
IF fbHttpGet.bError OR fbClient.bError THEN bError := TRUE; ELSE bError := FALSE; END_IF	
	hrErrorCode := fbClient.hrErrorCode;

END_FUNCTION_BLOCK

// ---- POUs/prgSmartMe.TcPOU
PROGRAM prgSmartMe
VAR
  fbSmartMe: FB_Get_Data_SmartMeApi_ElectricMeter; // 

  BilanzzaehlerKW                  : LREAL;  //{#lynus.ag#()}
  ProduktionPVAnlageKW             : LREAL;  //{#lynus.ag#()}
  TotalVerbraucherKW               : LREAL;  //{#lynus.ag#()}
  UVHalleNetzbauKW                 : LREAL;  //{#lynus.ag#()}
  UVGarderobentraktKW              : LREAL;  //{#lynus.ag#()}
  UVEKopfbauNordKW                 : LREAL;  //{#lynus.ag#()}
  UVSchulungsraumKW                : LREAL;  //{#lynus.ag#()}
  UVLadestationenKW                : LREAL;  //{#lynus.ag#()}
  UVErlebnisraumKW                 : LREAL;  //{#lynus.ag#()}
  UVMattenrainstrasse11AllgemeinKW : LREAL;  //{#lynus.ag#()}
  UVBueroKopfbauSuedKW             : LREAL;  //{#lynus.ag#()}
  UVMattenrainstrasse11HalleOstKW  : LREAL;  //{#lynus.ag#()}
  UVMattenrainstrasse11HalleWestKW : LREAL;  //{#lynus.ag#()}
  UVHeizungMattenrainstrasseKW     : LREAL;  //{#lynus.ag#()}
END_VAR

{region "Verbindung zu smart-me.com"}
  IF NOT fbSmartMe.bStart THEN
    // Init.
    fbSmartMe.sUsername    := 'ewsirnach'; 
    fbSmartMe.sPassword    := 'EWSirnach8370'; 
    fbSmartMe.tDelayRequest:= T#5S; 
    fbSmartMe.bStart       := TRUE;
  END_IF
  fbSmartMe();
{endregion}

IF NOT fbSmartMe.bValidResult THEN
  // Abbruch
  RETURN;
END_IF

BilanzzaehlerKW                  := fbSmartMe.arrListOfDevices[1].lrActivePower;
UVMattenrainstrasse11HalleWestKW := fbSmartMe.arrListOfDevices[2].lrActivePower;
UVMattenrainstrasse11HalleOstKW  := fbSmartMe.arrListOfDevices[3].lrActivePower;
UVHalleNetzbauKW                 := fbSmartMe.arrListOfDevices[4].lrActivePower;
UVHeizungMattenrainstrasseKW     := fbSmartMe.arrListOfDevices[5].lrActivePower;
ProduktionPVAnlageKW             := fbSmartMe.arrListOfDevices[6].lrActivePower;
UVGarderobentraktKW              := fbSmartMe.arrListOfDevices[7].lrActivePower;
UVEKopfbauNordKW                 := fbSmartMe.arrListOfDevices[8].lrActivePower;
UVBueroKopfbauSuedKW             := fbSmartMe.arrListOfDevices[9].lrActivePower;
UVSchulungsraumKW                := fbSmartMe.arrListOfDevices[10].lrActivePower;
UVLadestationenKW                := fbSmartMe.arrListOfDevices[11].lrActivePower;
UVErlebnisraumKW                 := fbSmartMe.arrListOfDevices[12].lrActivePower;
UVMattenrainstrasse11AllgemeinKW := fbSmartMe.arrListOfDevices[13].lrActivePower;
TotalVerbraucherKW               := fbSmartMe.arrListOfDevices[16].lrActivePower;

END_PROGRAM

// ---- POUs/prgHeizen.TcPOU
PROGRAM prgHeizen
VAR
  // Modbus Hoval
  fbHoval                     : FB_Hoval:= (CfgIpAddr:= '172.20.1.152');
  HalleMattenrain11Soll       : LREAL; //{#lynus.ag#()}
  HalleMattenrain11VLIst      : LREAL; //{#lynus.ag#()}
  RadGravierraumSoll          : LREAL; //{#lynus.ag#()}
  FbhGaderobeWCSoll           : LREAL; //{#lynus.ag#()}
  RadGravierraumIst           : LREAL; //{#lynus.ag#()}
  FbhGaderobeWCIst            : LREAL; //{#lynus.ag#()}
  LufterhitzerLagerSoll       : LREAL; //{#lynus.ag#()}
  BueroHusSoll                : LREAL; //{#lynus.ag#()}
  LufterhitzerLagerIst        : LREAL; //{#lynus.ag#()}
  BueroHusIst                 : LREAL; //{#lynus.ag#()}
  HalleMattenrain11Strategie  : INT;   //{#lynus.ag#()}
  RadGravierraumStrategie     : INT;   //{#lynus.ag#()}
  FbhGaderobeWCStrategie      : INT;   //{#lynus.ag#()}
  LufterhitzerLagerStrategie  : INT;   //{#lynus.ag#()}
  BueroHusStrategie           : INT;   //{#lynus.ag#()}


  //Temperatursensor OG1 Büro (Shelly)
  fbOG1BueroTemperatur  : FB_ShellyHT_Udp:= (Start:= TRUE, Port:= 50001);
	OG1BueroTemperatur		: LREAL;			//{#lynus.ag#()}
	OG1BueroFeuchte    		: LREAL;			//{#lynus.ag#()}
	OG1BueroBatterie   		: LREAL;			//{#lynus.ag#()}


END_VAR

{region "Hoval Heizung"}
  fbHoval(CfgIpAddr:= '172.20.1.152');
  HalleMattenrain11Soll       := fbHoval.HalleMattenrain11Soll;
  HalleMattenrain11VLIst      := fbHoval.HalleMattenrain11VLIst;
  RadGravierraumSoll          := fbHoval.RadGravierraumSoll;
  FbhGaderobeWCSoll           := fbHoval.FbhGaderobeWCSoll;
  RadGravierraumIst           := fbHoval.RadGravierraumIst;
  FbhGaderobeWCIst            := fbHoval.FbhGaderobeWCIst;
  LufterhitzerLagerSoll       := fbHoval.LufterhitzerLagerSoll;
  BueroHusSoll                := fbHoval.BueroHusSoll;
  LufterhitzerLagerIst        := fbHoval.LufterhitzerLagerIst;
  BueroHusIst                 := fbHoval.BueroHusIst;
  HalleMattenrain11Strategie  := fbHoval.HalleMattenrain11Strategie;
  RadGravierraumStrategie     := fbHoval.RadGravierraumStrategie;
  FbhGaderobeWCStrategie      := fbHoval.FbhGaderobeWCStrategie;
  LufterhitzerLagerStrategie  := fbHoval.LufterhitzerLagerStrategie;
  BueroHusStrategie           := fbHoval.BueroHusStrategie;
{endregion}

{region "Temperatursensor OG1 Büro (Shelly)"}
  fbOG1BueroTemperatur();

	OG1BueroTemperatur:= fbOG1BueroTemperatur.Temperatur;
	OG1BueroFeuchte   := fbOG1BueroTemperatur.Feuchte;
	OG1BueroBatterie  := fbOG1BueroTemperatur.Batterie;
{endregion}

END_PROGRAM

// ---- FB/FB_Hoval.TcPOU
FUNCTION_BLOCK FB_Hoval EXTENDS FbModbusTcpBase
// 07.05.2025 Elmar Vögel
VAR_INPUT
  END_VAR
VAR_OUTPUT
  HalleMattenrain11Soll       : LREAL;
  HalleMattenrain11VLIst      : LREAL;
  RadGravierraumSoll          : LREAL;
  FbhGaderobeWCSoll           : LREAL;
  RadGravierraumIst           : LREAL;
  FbhGaderobeWCIst            : LREAL;
  LufterhitzerLagerSoll       : LREAL;
  BueroHusSoll                : LREAL;
  LufterhitzerLagerIst        : LREAL;
  BueroHusIst                 : LREAL;
  HalleMattenrain11Strategie  : INT;
  RadGravierraumStrategie     : INT;
  FbhGaderobeWCStrategie      : INT;
  LufterhitzerLagerStrategie  : INT;
  BueroHusStrategie           : INT;
END_VAR

VAR CONSTANT
  cDelaySend : TIME:= T#1S;  
END_VAR

VAR
  iState      : INT;
  mPoll       : TON:= (PT:= T#1S);

  mReg        : ARRAY[0..10] OF WORD;
END_VAR

{region "Basis"}
  SUPER^();
{endregion}
{region "Modbus bearbeiten"}
  CASE iState OF
  0:  

    mPoll(IN:= TRUE);
    IF mPoll.Q THEN

      mPoll(IN:= FALSE);
  
      mCmd.UnitID   := 16#3;
      mCmd.Funktion := ModbusFunktion.ReadRegs;
      mCmd.MBAddr   := 16#06DC; // 1756
      mCmd.Quantity := 1; 
      mCmd.DatenAddr:= ADR(mReg);
      mCmd.DatenLen := SIZEOF(mReg);
  
      iState:= 100;
    END_IF

  100: SendNext(iState + 1);
  101:
    IF Empfang(cDelaySend) THEN

      IF NOT Error THEN
        HalleMattenrain11Soll:= TO_LREAL(mReg[0]) / 10.0;
      END_IF
         
      mCmd.UnitID   := 16#3;
      mCmd.Funktion := ModbusFunktion.ReadRegs;
      mCmd.MBAddr   := 16#06F3; // 1779
      mCmd.Quantity := 1; 
      mCmd.DatenAddr:= ADR(mReg);
      mCmd.DatenLen := SIZEOF(mReg);

      iState:= 110; 
    END_IF

  110: SendNext(iState + 1);
  111:
    IF Empfang(cDelaySend) THEN

      IF NOT Error THEN
        HalleMattenrain11VLIst:= TO_LREAL(mReg[0]) / 10.0;
      END_IF
         
      mCmd.UnitID   := 16#9;
      mCmd.Funktion := ModbusFunktion.ReadRegs;
      mCmd.MBAddr   := 16#1179; // 4473
      mCmd.Quantity := 2; 
      mCmd.DatenAddr:= ADR(mReg);
      mCmd.DatenLen := SIZEOF(mReg);

      iState:= 120; 
    END_IF

  120: SendNext(iState + 1);
  121:
    IF Empfang(cDelaySend) THEN

      IF NOT Error THEN
        RadGravierraumSoll:= TO_LREAL(mReg[0]) / 10.0;
        FbhGaderobeWCSoll := TO_LREAL(mReg[1]) / 10.0;
      END_IF
         
      mCmd.UnitID   := 16#9;
      mCmd.Funktion := ModbusFunktion.ReadRegs;
      mCmd.MBAddr   := 16#118A; // 4490
      mCmd.Quantity := 2; 
      mCmd.DatenAddr:= ADR(mReg);
      mCmd.DatenLen := SIZEOF(mReg);

      iState:= 130; 
    END_IF

  130: SendNext(iState + 1);
  131:
    IF Empfang(cDelaySend) THEN

      IF NOT Error THEN
        RadGravierraumIst:= TO_LREAL(mReg[0]) / 10.0;
        FbhGaderobeWCIst := TO_LREAL(mReg[1]) / 10.0;
      END_IF
         
      mCmd.UnitID   := 16#A;
      mCmd.Funktion := ModbusFunktion.ReadRegs;
      mCmd.MBAddr   := 16#11D7; // 4567
      mCmd.Quantity := 2; 
      mCmd.DatenAddr:= ADR(mReg);
      mCmd.DatenLen := SIZEOF(mReg);

      iState:= 140; 
    END_IF

  140: SendNext(iState + 1);
  141:
    IF Empfang(cDelaySend) THEN

      IF NOT Error THEN
        LufterhitzerLagerSoll:= TO_LREAL(mReg[0]) / 10.0;
        BueroHusSoll         := TO_LREAL(mReg[1]) / 10.0;
      END_IF
         
      mCmd.UnitID   := 16#A;
      mCmd.Funktion := ModbusFunktion.ReadRegs;
      mCmd.MBAddr   := 16#11E8; // 4584
      mCmd.Quantity := 2; 
      mCmd.DatenAddr:= ADR(mReg);
      mCmd.DatenLen := SIZEOF(mReg);

      iState:= 150; 
    END_IF

  150: SendNext(iState + 1);
  151:
    IF Empfang(cDelaySend) THEN

      IF NOT Error THEN
        LufterhitzerLagerIst:= TO_LREAL(mReg[0]) / 10.0;
        BueroHusIst         := TO_LREAL(mReg[1]) / 10.0;
      END_IF
         
      mCmd.UnitID   := 16#3;
      mCmd.Funktion := ModbusFunktion.ReadRegs;
      mCmd.MBAddr   := 16#6C02; // 27650
      mCmd.Quantity := 1; 
      mCmd.DatenAddr:= ADR(mReg);
      mCmd.DatenLen := SIZEOF(mReg);

      iState:= 160; 
    END_IF

  160: SendNext(iState + 1);
  161:
    IF Empfang(cDelaySend) THEN

      IF NOT Error THEN
        HalleMattenrain11Strategie:= TO_INT(mReg[0]);
      END_IF
         
      mCmd.UnitID   := 16#9;
      mCmd.Funktion := ModbusFunktion.ReadRegs;
      mCmd.MBAddr   := 16#78BB; // 30907
      mCmd.Quantity := 2; 
      mCmd.DatenAddr:= ADR(mReg);
      mCmd.DatenLen := SIZEOF(mReg);

      iState:= 170; 
    END_IF

  170: SendNext(iState + 1);
  171:
    IF Empfang(cDelaySend) THEN

      IF NOT Error THEN
        RadGravierraumStrategie:= TO_INT(mReg[0]);
        FbhGaderobeWCStrategie := TO_INT(mReg[1]);
      END_IF
         
      mCmd.UnitID   := 16#A;
      mCmd.Funktion := ModbusFunktion.ReadRegs;
      mCmd.MBAddr   := 16#78BE; // 30910
      mCmd.Quantity := 2; 
      mCmd.DatenAddr:= ADR(mReg);
      mCmd.DatenLen := SIZEOF(mReg);

      iState:= 180; 
    END_IF

  180: SendNext(iState + 1);
  181:
    IF Empfang(cDelaySend) THEN

      IF NOT Error THEN
        LufterhitzerLagerStrategie:= TO_INT(mReg[0]);
        BueroHusStrategie         := TO_INT(mReg[1]);
      END_IF
         
      iState:= 800; 
    END_IF

  800:
    // Fertig
    iState:= 0;
  END_CASE
{endregion}

METHOD PRIVATE SendNext : BOOL
VAR_INPUT
  StepNext : INT;
END_VAR

  SendNext:= FALSE;
  IF SUPER^.Send() THEN

    iState:= StepNext;
    SendNext:= TRUE;
  END_IF
END_METHOD

END_FUNCTION_BLOCK

// ---- FB/FB_ShellyHT_Udp.TcPOU
FUNCTION_BLOCK FB_ShellyHT_Udp
// 14.02.2025 Elmar Vögel
VAR_INPUT
  Start : BOOL;         // Kommunikation aktivieren
  Port  : UINT:= 50001; // Tcp Port
END_VAR
VAR_OUTPUT PERSISTENT
  Temperatur   : LREAL;        // Istwerte
  Feuchte      : LREAL;
  Batterie     : LREAL;
  Geraet       : T_MaxString;
END_VAR
VAR_OUTPUT
  Bereit       : BOOL;        // Info
  SocketState  : E_SocketConnectionlessState;
  RecCount     : UINT;  
END_VAR

VAR
  fbSocket  : FB_ConnectionlessSocket;
  fbReceive : FB_SocketUdpReceiveFrom;
  sReceive  : STRING(2000);
  fbRecTon  : TON;
END_VAR

{region "Init. Socket öffnen"}
  IF Start AND NOT fbSocket.bEnable THEN
    // Trig. Konfiguraton
    fbSocket.nMode     := CONNECT_MODE_ENABLEDBG;
    fbSocket.tReconnect:= T#60S;
    
    fbRecTon.PT:= T#100MS;
  END_IF

  fbSocket(
    nLocalPort:= Port, 
    bEnable   := Start, 
    eState    => SocketState);
{endregion}

{region "Daten lesen"}
  fbRecTon(IN:=  NOT fbReceive.bBusy);
  IF fbRecTon.Q THEN
  
    fbReceive.bExecute:= TRUE;
    fbRecTon(IN:= FALSE);
  END_IF
  
  fbReceive(
    sSrvNetId:= , 
    hSocket  := fbSocket.hSocket, 
    cbLen    := SIZEOF(sReceive), 
    pDest    := ADR(sReceive));
  
  IF fbReceive.bExecute AND NOT fbReceive.bBusy THEN
    
    Bereit:= NOT fbReceive.bError;
    fbReceive.bExecute:= FALSE;
    IF fbReceive.nRecBytes > 0 THEN

      ConvertData();
      RecCount:= RecCount + 1;
    END_IF
  END_IF  

  IF NOT Start THEN  

    Bereit:= FALSE;
  END_IF
{endregion}

METHOD PRIVATE ConvertData
VAR_INST
  fbJson      : FB_JsonDomParser;
	jsonDoc		  : SJsonValue;
	jsonParams	: SJsonValue;
	jsonProp	  : SJsonValue;
	jsonValue	  : SJsonValue;
END_VAR
(* JSON
{
   "src":"shellyhtg3-8cbfea9a98d4",
   "dst":"UDP_out",
   "method":"NotifyFullStatus",
   "params":{
      "ts":1739462691.05,
      "ble":{
         
      },
      "cloud":{
         "connected":false
      },
      "devicepower:0":{
         "id":0,
         "battery":{
            "V":5.87,
            "percent":93
         },
         "external":{
            "present":false
         }
      },
      "ht_ui":{
         
      },
      "humidity:0":{
         "id":0,
         "rh":42.7
      },
      "mqtt":{
         "connected":false
      },
      "sys":{
         "mac":"8CBFEA9A98D4",
         "restart_required":false,
         "time":null,
         "unixtime":null,
         "uptime":0,
         "ram_size":255900,
         "ram_free":165324,
         "fs_size":1048576,
         "fs_free":745472,
         "cfg_rev":55,
         "kvs_rev":0,
         "webhook_rev":0,
         "available_updates":{
            
         },
         "wakeup_reason":{
            "boot":"deepsleep_wake",
            "cause":"button"
         },
         "wakeup_period":7200,
         "reset_reason":8
      },
      "temperature:0":{
         "id":0,
         "tC":21.3,
         "tF":70.4
      },
      "wifi":{
         "sta_ip":"192.168.66.90",
         "status":"got ip",
         "ssid":"VSA",
         "rssi":-59
      },
      "ws":{
         "connected":false
      }
   }
}
*)

  jsonDoc := fbJson.ParseDocument(sReceive);
  MEMSET(ADR(sReceive), 0, SIZEOF(sReceive));

  IF (jsonValue:= fbJson.FindMember(jsonDoc, 'src')) <> 0 THEN
    Geraet:= fbJson.GetString(jsonValue);
  END_IF  

  IF (jsonParams:= fbJson.FindMember(jsonDoc, 'params')) <> 0 THEN

    IF (jsonProp:= fbJson.FindMember(jsonParams, 'temperature:0')) <> 0 THEN
      IF (jsonValue:= fbJson.FindMember(jsonProp, 'tC')) <> 0 THEN
        Temperatur:= fbJson.GetDouble(jsonValue);
      END_IF
    END_IF

    IF (jsonProp:= fbJson.FindMember(jsonParams, 'humidity:0')) <> 0 THEN
      IF (jsonValue:= fbJson.FindMember(jsonProp, 'rh')) <> 0 THEN
        Feuchte:= fbJson.GetDouble(jsonValue);
      END_IF
    END_IF

    IF (jsonProp:= fbJson.FindMember(jsonParams, 'devicepower:0')) <> 0 THEN
      IF (jsonProp:= fbJson.FindMember(jsonProp, 'battery')) <> 0 THEN
        IF (jsonValue:= fbJson.FindMember(jsonProp, 'percent')) <> 0 THEN
          Batterie:= fbJson.GetDouble(jsonValue);
        END_IF
      END_IF  
    END_IF
  END_IF
END_METHOD

END_FUNCTION_BLOCK

// ---- POUs/prgComEffIO.TcPOU
PROGRAM prgComEffIO
VAR
	fbCom		: FB_MqttCommunicator_V5;
END_VAR

// CX-7BDACD
fbCom(
	bConnect:= TRUE, 
	strAuthKey := 'ENE87365342998',
	sUserName:= '8be10145-b694-4bbc-810e-ed40ca315ba9', 
	sUserPassword:= '78d23592-454c-40a8-9e0a-2748027b0c68', 
	eSavePositionCertificate:= eSavePositionOnPLC.ePostionHardDisk,
	time_HeartBeat_sec:= T#50S, 
	bConnected=> , 
	bError=> , 
	hrErrorCode=> , 
	eConnectionState=> , 
	eErrorMessage_Out=> );

END_PROGRAM

// ---- FB/FB_Shelly_HT.TcPOU
FUNCTION_BLOCK FB_Shelly_HT
VAR_INPUT
	bStart				: BOOL;
	tDelayRequest		: TIME;		//Timer for delay before start with the next read or write Request
	sHostname			: STRING(255);		//Hostname or IP Adress from the Server
END_VAR

VAR_IN_OUT
END_VAR

VAR_OUTPUT
	bValidResult		: BOOL;							//Valid Result received from Server
    bBusy				: BOOL;							//Function is Busy
    bError				: BOOL;							//Error sucess
	bDone				: BOOL;							//True after the decoding from the received Json File
	bConnected			: BOOL;							//Connection to the Server
	lr_Temperature		: LREAL;						//Received Value
	lr_Humidity			: LREAL;
	hrErrorCode       	: HRESULT;						//Error Result from Http Client
END_VAR

VAR
	fbClient			: FB_IotHttpClient;
	fbHttpGet			: FB_Shelly_HT_Helper;
	timStartRequest		: TON;							//Timer to Start the Request
	FPStartRequest		: R_TRIG;						//Internal positive Edge
	FPDone				: R_TRIG;						//Internal positive Edge
	FNStart				: F_TRIG;						//Internal negative Edge
	y: INT;
END_VAR

(*------------------------------------------------------------------------------------Configure HTTP Client------------------------------------------------------------------------------------------------------*)

fbClient.sHostName := sHostname;
fbClient.tConnectionTimeout := T#30S;

IF NOT fbClient.bConfigured THEN 
	fbClient.nHostPort:= 80;
	fbClient.bKeepAlive := TRUE;
	fbClient.tConnectionTimeout := T#30S;
END_IF


//Timer to start the Request
FPStartRequest(CLK:= bStart, Q=> );
timStartRequest(IN:= fbClient.bConfigured AND bStart AND NOT timStartRequest.Q, PT:= tDelayRequest, Q=> , ET=> );

IF ((timStartRequest.Q AND NOT bBusy) OR (FPStartRequest.Q AND NOT bBusy AND fbClient.bConfigured)) THEN 
	y:=y+1;
	fbHttpGet.bSend := TRUE; 
END_IF

				
//Http Get Function

fbHttpGet(
	bSend:= , 
	fbClient:= , 
	bBusy=> , 
	bError=> , 
	lr_Temperature=> lr_Temperature, 
	lr_Humidity=> lr_Humidity,
	bSend:= , 
	fbClient:= fbClient, 
	bBusy=> bBusy, 
	bError=> ,
	sContentStatus=> ,
	sContentM0=> ,
	sContentM1=> ,
	sContentM2=> );
	



fbHttpGet.bSend := FALSE;

FPDone(CLK:= bDone, Q=> );

(*
//Http Client
FNStart(CLK:= bStart, Q=> );
	IF FNStart.Q THEN fbClient.Disconnect(); END_IF
*)

fbClient.Execute();

//Error
IF fbHttpGet.bError OR fbClient.bError THEN 
	bError := TRUE; 
ELSE 
	bError := FALSE; 
END_IF	

hrErrorCode := fbClient.hrErrorCode;

END_FUNCTION_BLOCK

// ---- FB/FB_Shelly_HTplus.TcPOU
FUNCTION_BLOCK FB_Shelly_HTplus
VAR_INPUT
	bStart				: BOOL;
	tDelayRequest		: TIME;		//Timer for delay before start with the next read or write Request
	sHostname			: STRING(255);		//Hostname or IP Adress from the Server
END_VAR

VAR_IN_OUT
END_VAR

VAR_OUTPUT
	bValidResult		: BOOL;							//Valid Result received from Server
    bBusy				: BOOL;							//Function is Busy
    bError				: BOOL;							//Error sucess
	bDone				: BOOL;							//True after the decoding from the received Json File
	bConnected			: BOOL;							//Connection to the Server
	lr_Temperature		: LREAL;						//Received Value
	lr_Humidity			: LREAL;
	hrErrorCode       	: HRESULT;						//Error Result from Http Client
END_VAR

VAR
	fbClient			: FB_IotHttpClient;
	fbHttpGet			: FB_Shelly_HTplus_Helper;
	timStartRequest		: TON;							//Timer to Start the Request
	FPStartRequest		: R_TRIG;						//Internal positive Edge
	FPDone				: R_TRIG;						//Internal positive Edge
	FNStart				: F_TRIG;						//Internal negative Edge
	y: INT;
END_VAR

(*------------------------------------------------------------------------------------Configure HTTP Client------------------------------------------------------------------------------------------------------*)

fbClient.sHostName := sHostname;
fbClient.tConnectionTimeout := T#30S;

IF NOT fbClient.bConfigured THEN 
	fbClient.nHostPort:= 80;
	fbClient.bKeepAlive := TRUE;
	fbClient.tConnectionTimeout := T#30S;
END_IF


//Timer to start the Request
FPStartRequest(CLK:= bStart, Q=> );
timStartRequest(IN:= fbClient.bConfigured AND bStart AND NOT timStartRequest.Q, PT:= tDelayRequest, Q=> , ET=> );

IF ((timStartRequest.Q AND NOT bBusy) OR (FPStartRequest.Q AND NOT bBusy AND fbClient.bConfigured)) THEN 
	y:=y+1;
	fbHttpGet.bSend := TRUE; 
END_IF

				
//Http Get Function

fbHttpGet(
	bSend:= , 
	fbClient:= , 
	bBusy=> , 
	bError=> , 
	lr_Temperature=> lr_Temperature, 
	lr_Humidity=> lr_Humidity,
	bSend:= , 
	fbClient:= fbClient, 
	bBusy=> bBusy, 
	bError=> ,
	sContentStatus=> ,
	sContentM0=> ,
	sContentM1=> ,
	sContentM2=> );
	



fbHttpGet.bSend := FALSE;

FPDone(CLK:= bDone, Q=> );

(*
//Http Client
FNStart(CLK:= bStart, Q=> );
	IF FNStart.Q THEN fbClient.Disconnect(); END_IF
*)

fbClient.Execute();

//Error
IF fbHttpGet.bError OR fbClient.bError THEN 
	bError := TRUE; 
ELSE 
	bError := FALSE; 
END_IF	

hrErrorCode := fbClient.hrErrorCode;

END_FUNCTION_BLOCK

// ---- FB/FB_Shelly_HTplus_Helper.TcPOU
FUNCTION_BLOCK FB_Shelly_HTplus_Helper
VAR_INPUT
	bSend				: BOOL;
END_VAR

VAR_IN_OUT
	fbClient			: FB_IotHttpClient;
END_VAR

VAR_OUTPUT
	bBusy				: BOOL;
	bError				: BOOL;
	lr_Temperature		: LREAL;						//Received Value
	lr_Humidity			: LREAL;
END_VAR

VAR
	fbRequestStatus		: FB_IotHttpRequest;
	fbJson				: FB_JsonDomParser;
	nState				: UDINT;
	RisingEdge			: R_TRIG;
	timTimeout			: TON;
	tTimeOut			: TIME := T#50S;
	bGetContentResult	: BOOL;
	sContentStatus		: STRING(511);
	sContentM0			: STRING(511);
	sContentM1			: STRING(511);
	sContentM2			: STRING(511);
	
	bGetJsonResult		: BOOL;
	jsonDoc				: SJsonValue;
	jsonVal				: SJsonValue;
	
	nReqCount			: UDINT;	
	nResCount			: UDINT;
	nValidResCount		: UDINT;
	nErrCount			: UDINT;
	x: INT;
END_VAR

//Timer for Timeout
timTimeout(IN:= nState = 1 AND bBusy, PT:= tTimeOut, Q=> , ET=> );
	IF timTimeout.Q THEN 
		nState := 0;
		bBusy := FALSE;
	END_IF

RisingEdge(CLK:= bSend );
CASE nState OF
0:	
	IF RisingEdge.Q THEN 
		IF 
			fbRequestStatus.SendRequest(sUri:='/rpc/Humidity.GetStatus?id=0', fbClient:=fbClient, eRequestType:=ETcIotHttpRequestType.HTTP_Get, 0, 0, 0) THEN				
			nState:= 1;
			nReqCount:= nReqCount+1;
			bBusy:= TRUE;
			bError:= FALSE;
		END_IF					
	END_IF
1:
	x:=x+1;
	IF  NOT fbRequestStatus.bBusy THEN
		bError:= TRUE;
			
		IF NOT fbRequestStatus.bError THEN				 
			bGetContentResult:= fbRequestStatus.GetContent(pContent:= ADR(sContentStatus), nContentSize:= SIZEOF(sContentStatus), bSetNullTermination:= TRUE);
			IF fbRequestStatus.nStatusCode >= 200 AND fbRequestStatus.nStatusCode < 300 THEN
				bGetJsonResult:= FALSE;
				jsonDoc:= fbRequestStatus.GetJsonDomContent(fbJson);
				IF jsonDoc <> 0 THEN
					bGetJsonResult:= TRUE;
					IF fbJson.HasMember(jsonDoc, 'tC')  THEN
						jsonVal:= fbJson.FindMember(jsonDoc, 'tC');
						nValidResCount:= nValidResCount+1;
						IF fbJson.IsDouble(jsonVal) THEN							
							lr_Temperature:= fbJson.GetDouble(jsonVal);									
						END_IF
						bError:= FALSE;
					END_IF
				END_IF
				nResCount:= nResCount+1;			
			END_IF
		END_IF
		
		nState:= 0;
		bBusy:= FALSE;
		IF bError THEN
			nErrCount:= nErrCount+1;
		END_IF
	END_IF  	
END_CASE

END_FUNCTION_BLOCK

// ---- FB/FB_Shelly_Pro.TcPOU
FUNCTION_BLOCK FB_Shelly_Pro1PM
VAR_INPUT
	bStart				: BOOL;
	tDelayRequest		: TIME;				//Timer for delay before start with the next read or write Request
	sHostname			: STRING(255);		//Hostname or IP Adress from the Server
	//bOnP1				: BOOL;
	//bOffP1				: BOOL;
	//bEnableControl		: BOOL;
END_VAR

VAR_OUTPUT
	bValidResult				: BOOL;															//Valid Result received from Server
    bBusy						: BOOL;															//Function is Busy
    bError						: BOOL;															//Error sucess
	bDone						: BOOL;															//True after the decoding from the received Json File
	bConnected					: BOOL;															//Connection to the Server
	hrErrorCode       			: HRESULT;														//Error Result from Http Client
	lrpowerP1					: LREAL;														//Received Value
	lrvoltageP1					: LREAL;														//Received Value
	lrenergyP1					: LREAL;														//Received Value
	lrTemperatureP1				: LREAL;														//Received Value
	bStateP1					: BOOL;
END_VAR

VAR
	fbClient					: FB_IotHttpClient;
	fbHttpGet					: FB_Shelly_Pro1PM_Helper;
	timStartRequest				: TON;															//Timer to Start the Request
	FPStartRequest				: R_TRIG;														//Internal positive Edge
	FPDone						: R_TRIG;														//Internal positive Edge
	FNStart						: F_TRIG;														//Internal negative Edge
	(* There are no Switches 
	SwitchOnP1					: R_TRIG;
	SwitchOffP1					: R_TRIG;
	rs_Switch_ON: Rs;
	rs_Switch_OFF: RS;
	*) 
	x: INT;
END_VAR

bError := FALSE;
(*------------------------------------------------------------------------------------Configure HTTP Client------------------------------------------------------------------------------------------------------*)

fbClient.sHostName := sHostname;
fbClient.tConnectionTimeout := T#25S;

IF NOT fbClient.bConfigured THEN 
	fbClient.nHostPort:= 80;
	fbClient.bKeepAlive := TRUE;
	fbClient.tConnectionTimeout := T#25S;
END_IF


//Timer to start the Request
FPStartRequest(CLK:= bStart, Q=> );
timStartRequest(	IN:= fbClient.bConfigured AND bStart AND NOT timStartRequest.Q, 
					PT:= tDelayRequest, 
					Q=> , 
					ET=> );
IF ((timStartRequest.Q AND NOT bBusy) OR (FPStartRequest.Q AND NOT bBusy AND fbClient.bConfigured)) THEN 
	fbHttpGet.bSend := TRUE; 
	x:=x+1;
END_IF

				
//Http Get Function
fbHttpGet(
	lrapowerP1 => lrpowerP1, 
	lrvoltageP1 => lrvoltageP1, 
	lraenergyP1 => lrenergyP1,
	lrTemperatureP1 => lrTemperatureP1,
	bSend:= , 
	fbClient:= fbClient, 
	bBusy=> bBusy, 
	bError=> ,
	sContentS0=> ,
	bStateP1=>bStateP1 );


fbHttpGet.bSend := FALSE;

FPDone(CLK:= bDone, Q=> );

// zum testen ob dadurch die verbindung aufrechtbleibt nach dem schalten 
// --> error geht nicht mehr low!
// IF NOT bError  THEN
	fbClient.Execute();
// ELSE
//	fbClient.Disconnect();
// END_IF

//Error
IF fbHttpGet.bError OR fbClient.bError THEN bError := TRUE; ELSE bError := FALSE; END_IF	
	hrErrorCode := fbClient.hrErrorCode;
	
(*
// Relay Control, Switch P1
SwitchOnP1(CLK:=bOnP1);
rs_Switch_ON(	Set:= SwitchOnP1.Q AND bEnableControl,
				Reset1 := bStateP1);	// OR fbHttpGet.timTimeoutSwitch.Q);
				
IF rs_Switch_ON.Q1 AND bEnableControl THEN
	fbHttpGet.bSetOnP1 := TRUE;
ELSE
	fbHttpGet.bSetOnP1 := FALSE;
END_IF

SwitchOffP1(CLK:=bOffP1);
rs_Switch_OFF(	Set:= SwitchOffP1.Q AND bEnableControl,
				Reset1 := NOT bStateP1);	// OR fbHttpGet.timTimeoutSwitch.Q);
				
IF rs_Switch_OFF.Q1 AND bEnableControl THEN
	fbHttpGet.bSetOffP1 := TRUE;
ELSE
	fbHttpGet.bSetOffP1 := FALSE;
END_IF
*)

END_FUNCTION_BLOCK
